PROGRAM P_RecipeChange
VAR
	b_recipe_bool_change :R_trig;
	b_recipe_real_change :R_trig;
	b_recipe_was_changed_real :BOOL;
	b_recipe_was_changed_bool :BOOL;
	lr_old_param_bool :LREAL;
	lr_new_param_bool :LREAL;
	i :INT;
	nIndex      : INT := 0; 
    nTotalItems : INT := 500; 
	b_clear_recipe_history :BOOL:=FALSE;
END_VAR

b_recipe_bool_change(clk:= gvl_recipe.b_recipe_bool_change);
b_recipe_real_change(clk:= gvl_recipe.b_recipe_real_change);
b_clear_recipe_history:=FALSE;
IF gvl_recipe.b_recipe_real_change THEN //zmiana real
	IF (gvl_recipe.lr_recipe_change<>gvl_recipe.lr_recipe_change_1)  THEN
		b_recipe_was_changed_real:=TRUE;				
	END_IF
ELSE
	IF  gvl_recipe.b_recipe_bool_change THEN
			b_recipe_was_changed_bool:=TRUE;		
			IF gvl_recipe.s_recupe_change_4="false" THEN
				lr_old_param_bool:=0;
				lr_new_param_bool:=1;
			END_IF
			IF gvl_recipe.s_recupe_change_4="true" THEN
				lr_old_param_bool:=1;
				lr_new_param_bool:=0;
			END_IF
		//END_IF		
	END_IF
END_IF

IF b_recipe_bool_change.q OR b_recipe_real_change.q THEN
	FOR i := 499 TO 1 BY -1 DO
		gvl_recipe.ArRecipeChanges[i].old_value:=gvl_recipe.ArRecipeChanges[i-1].old_value;
		gvl_recipe.ArRecipeChanges[i].new_value:=gvl_recipe.ArRecipeChanges[i-1].new_value;
		gvl_recipe.ArRecipeChanges[i].when_changed:=gvl_recipe.ArRecipeChanges[i-1].when_changed;
		gvl_recipe.ArRecipeChanges[i].who_changed:=gvl_recipe.ArRecipeChanges[i-1].who_changed;
		gvl_recipe.ArRecipeChanges[i].which_param_name:=gvl_recipe.ArRecipeChanges[i-1].which_param_name;
		gvl_recipe.ArRecipeChanges[i].which_param_var:=gvl_recipe.ArRecipeChanges[i-1].which_param_var;
		gvl_recipe.ArRecipeChanges[i].which_param_cntr:=gvl_recipe.ArRecipeChanges[i-1].which_param_cntr;
		gvl_recipe.ArRecipeChanges[i].which_recipe:=gvl_recipe.ArRecipeChanges[i-1].which_recipe;
	END_FOR
END_IF
IF b_recipe_was_changed_real THEN
		gvl_recipe.ArRecipeChanges[0].old_value:=gvl_recipe.lr_recipe_change;
		gvl_recipe.ArRecipeChanges[0].new_value:=gvl_recipe.lr_recipe_change_1;
		gvl_recipe.ArRecipeChanges[0].when_changed:=P_time.actual_date_meawhile;
		gvl_recipe.ArRecipeChanges[0].who_changed:=gvl_recipe.s_recipe_change;
		gvl_recipe.ArRecipeChanges[0].which_param_name:=gvl_recipe.s_recipe_change_1;
		gvl_recipe.ArRecipeChanges[0].which_param_var:=wconcat(" '' ",gvl_recipe.s_recipe_change_2);
		gvl_recipe.ArRecipeChanges[0].which_param_cntr:=Wconcat("'",gvl_recipe.s_recipe_change_3);
		gvl_recipe.ArRecipeChanges[0].which_param_cntr:=Wconcat(gvl_recipe.ArRecipeChanges[0].which_param_cntr,"'");
		gvl_recipe.ArRecipeChanges[0].which_recipe:=gvl_recipe.s_recipe_name;
	END_IF
IF b_recipe_was_changed_bool THEN
		gvl_recipe.ArRecipeChanges[0].old_value:=lr_old_param_bool;
		gvl_recipe.ArRecipeChanges[0].new_value:=lr_new_param_bool;
		gvl_recipe.ArRecipeChanges[0].when_changed:=P_time.actual_date_meawhile;
		gvl_recipe.ArRecipeChanges[0].who_changed:=gvl_recipe.s_recipe_change;
		gvl_recipe.ArRecipeChanges[0].which_param_name:=gvl_recipe.s_recipe_change_1;
		gvl_recipe.ArRecipeChanges[0].which_param_var:=wconcat(" '' ",gvl_recipe.s_recipe_change_2);
		gvl_recipe.ArRecipeChanges[0].which_param_cntr:=Wconcat("'",gvl_recipe.s_recipe_change_3);
		gvl_recipe.ArRecipeChanges[0].which_param_cntr:=Wconcat(gvl_recipe.ArRecipeChanges[0].which_param_cntr,"'");
		gvl_recipe.ArRecipeChanges[0].which_recipe:=gvl_recipe.s_recipe_name;
END_IF

IF b_clear_recipe_history OR gvl_recipe.b_recipe_changes_clear THEN
	p_arraytofile.nFileCounter:=1;
FOR nIndex := 0 TO nTotalItems DO
    gvl_Recipe.ArRecipeChanges[nIndex].old_value := 0.0;
    gvl_Recipe.ArRecipeChanges[nIndex].new_value := 0.0;
    gvl_Recipe.ArRecipeChanges[nIndex].who_changed := "";         // WSTRING pusty
    gvl_Recipe.ArRecipeChanges[nIndex].when_changed := DT#1970-01-01-00:00:00; // Wartość domyślna dla DT
    gvl_Recipe.ArRecipeChanges[nIndex].which_param_name := "";     // WSTRING pusty
    gvl_Recipe.ArRecipeChanges[nIndex].which_param_var := "";      // WSTRING pusty
	gvl_recipe.ArRecipeChanges[nIndex].which_param_cntr:="";
	gvl_recipe.ArRecipeChanges[nIndex].which_recipe:="";
END_FOR
END_IF

IF gvl_recipe.ArRecipeChanges[400].which_param_cntr<>"" THEN
	b_clear_recipe_history:=TRUE;	
END_IF
		
IF gvl_recipe.b_recipe_bool_change=FALSE THEN
	b_recipe_was_changed_bool:=FALSE;
END_IF

IF gvl_recipe.b_recipe_real_change=FALSE THEN
		b_recipe_was_changed_real:=FALSE;
END_IF

END_PROGRAM

(* stored: Version 1.1.0.1, ProductVersion 3.1.4026.13, FileIdentifier 280337a3ef72003144a8b6c00c0e53c39b74da63, FileSignature 9d4fd9eaff41b13b9f273dc46a90c4ecf12062ff04b6fa29958b219992202f4712701032e9664c612f8d6132d72ba59520be7f6423b1dd877c816952464716e1bfe4101f343e8e5d4acb4ccdc768d63ff15720947f3f15e3a60f021ce318e69fe01bb10f2041652da1a974d1a34f23544b91b823c4771cdbcb4563bcc062274c1824cbd2045eb865aac0296b895b91edc4fca12c1770990e63ddb616cba76418d0ffa9019ccae0eec60aec76ec3dc594999a64a72abc32ff153ad1f6f74eb0975f33f21454e5358869cc4ec6b779a917a040813b4ab7809c8fe6ead578f8c1b21172d9f7367ccf627b9d400c75d06c3181314ad7e772a35a85d214ef1175ca9e
   POU P_RecipeChange: Id {1b566b17-25b1-4b47-934c-7c4e3bb9ab3a}, SpecialFunc None *)
